Universal Robots PolyScope program: place_stick.urp

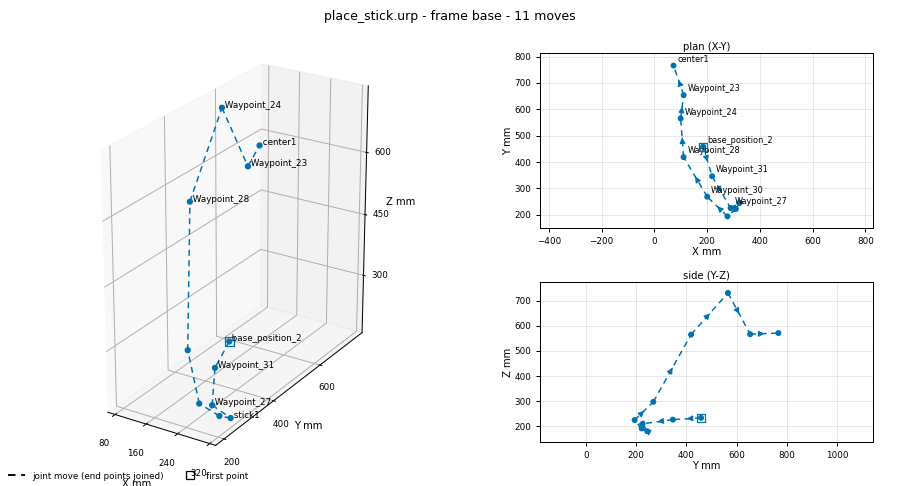
[picture p0: tool path of place_stick.urp in frame base, 11 of 11 moves have a stored position in this frame; points joined in program order, loops and branches not executed]
Program place_stick (installation=default directory=/programs/Nicolas Arteaga createdIn=5.12.4.1101661 lastSavedIn=5.12.4.1101661 robotSerialNumber=20225502378)
Calibrated DH parameters: a=[0.00022, -0.425328, -0.389701, 0.000059, 0.000065, 0]; d=[0.162608, 0.803456, 9.992211, -10.662202, 0.099702, 0.099559]; alpha=[1.570756, 0.001543, 0.004316, 1.570651, -1.570122, 0]; deltaTheta=[0, 0.002917, 0.116094, -0.119008, 0, -0.000001]
Robot Program (runOnlyOnce=true)
  'Takes the first wood stick and places it in the center of the cotton candy machine'
  MoveJ speed 60 deg/s, acceleration 80 deg/s^2 (useActiveTCP=true) feature=Base
    Waypoint base_position_2: TCP in base x=184.715 y=458.614 z=234.006 mm, rx=-1.6866 ry=-0.757 rz=-1.7388 rad; joints [237.954, -104.402, 143.977, -41.546, 99.477, 90] deg; TCP offset x=0 y=0 z=191.5 mm, rx=0 ry=0 rz=0 rad
    URCap Gripper Activate (Robotiq_Grippers, Robotiq Inc.) dataModel(ResetAndActivateKey=false)
    URCap Gripper (Robotiq_Grippers, Robotiq Inc.) dataModel(position=70.0, force=0.0, speed=100.0, positionInDouble=70.0, forceInDouble=0.0, speedInDouble=100.0, slaveIds=[9], blocking=true)
    Waypoint Waypoint_31: TCP in base x=219.073 y=346.37 z=226.939 mm, rx=-1.0793 ry=1.1503 rz=-0.4496 rad; joints [242.985, -108.839, 146.791, -38.8, 126.314, 210] deg; TCP offset x=0 y=0 z=191.5 mm, rx=0 ry=0 rz=0 rad
    Waypoint Waypoint_27: TCP in base x=288.911 y=225.994 z=210.348 mm, rx=-0.5682 ry=1.4712 rz=-0.493 rad; joints [230.777, -108.395, 149.908, -42.839, 137.738, 230] deg; TCP offset x=0 y=0 z=191.5 mm, rx=0 ry=0 rz=0 rad
    Waypoint stick1: TCP in base x=322.798 y=244.707 z=180.935 mm, rx=-0.6006 ry=1.5021 rz=-0.5325 rad; joints [227.883, -97.858, 147.006, -47.332, 135.838, 229.943] deg; TCP offset x=0 y=0 z=191.5 mm, rx=0 ry=0 rz=0 rad
    URCap Gripper (Robotiq_Grippers, Robotiq Inc.) dataModel(position=100.0, force=0.0, speed=0.0, positionInDouble=100.0, forceInDouble=0.0, speedInDouble=0.0, slaveIds=[9], blocking=true)
    Waypoint Waypoint_3: TCP in base x=308.934 y=222.719 z=191.895 mm, rx=-0.6005 ry=1.5021 rz=-0.5324 rad; joints [226.032, -105.235, 149.7, -42.849, 134.017, 229.721] deg
    Waypoint Waypoint_4: TCP in base x=277.219 y=194.361 z=225.221 mm, rx=-0.5767 ry=1.5048 rz=-0.5799 rad; joints [231.096, -114.882, 148.99, -33.185, 141.571, 228.474] deg
    Waypoint Waypoint_30: TCP in base x=200.562 y=268.796 z=297.612 mm, rx=-1.3009 ry=0.8471 rz=-0.8634 rad; joints [232.325, -138.788, 148.891, -15.287, 116.251, 180] deg; TCP offset x=0 y=0 z=191.5 mm, rx=0 ry=0 rz=0 rad
    Waypoint Waypoint_28: TCP in base x=110.872 y=418.885 z=565.169 mm, rx=-1.6121 ry=0.3611 rz=-0.2078 rad; joints [200.913, -129.115, 99.418, 36.172, 41.428, 180] deg; TCP offset x=0 y=0 z=191.5 mm, rx=0 ry=0 rz=0 rad
    Waypoint Waypoint_24: TCP in base x=99.712 y=565.5 z=730.734 mm, rx=-1.4619 ry=0.2517 rz=-0.2966 rad; joints [243.031, -99.822, 65.521, 28.761, 83.192, 180] deg; TCP offset x=0 y=0 z=191.5 mm, rx=0 ry=0 rz=0 rad
    Waypoint Waypoint_23: TCP in base x=111.331 y=653.695 z=566.749 mm, rx=-1.7943 ry=0.2693 rz=-0.1351 rad; joints [243.037, -87.632, 65.808, 35.91, 77.265, 180] deg; TCP offset x=0 y=0 z=191.5 mm, rx=0 ry=0 rz=0 rad
    Waypoint center1: TCP in base x=72.723 y=766.045 z=571.175 mm, rx=-1.5688 ry=-0.0203 rz=0.0146 rad; joints [244.553, -79.065, 65.7, 13.074, 63.165, 180.144] deg; TCP offset x=0 y=0 z=191.5 mm, rx=0 ry=0 rz=0 rad
